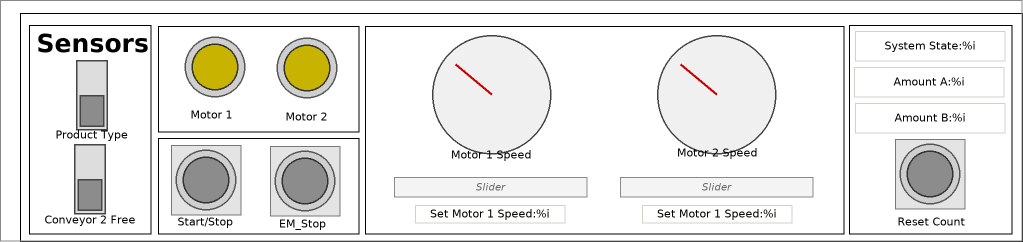
VISUALIZATION Visualization  // 1023x242
    Rectangle (20,13 1003x229)
    Rectangle (849,25 163x209)
    Rectangle (158,138 201x96)
    Rectangle (365,26 479x208)
    Rectangle (158,26 201x106)
    Rectangle (29,25 122x209)
    Lamp1 (180,32 70x70), style: Lamp-Lamp1-Yellow
    Lamp1 (272,33 70x70), variable: GVL.Motor2_State, style: Lamp-Lamp1-Yellow
    DipSwitch (57,60 70x70), variable: GVL.SensorInput, behaviour: TOGGLE, style: Switch-DipSwitch-Gray
    DipSwitch (55,144 70x70), variable: GVL.Conveyor2_Free, behaviour: TOGGLE, style: Switch-DipSwitch-Gray
    Label (18,28 150x30), "Sensors"
    Label (176,100 71x30), "Motor 1"
    Label (271,102 71x30), "Motor 2"
    Meter180 (386,35 211x119), value: GVL.CurrentMotor1_Speed, style: Meter-Meter180-Gray, scale format: %.1f, scale 0..100
    Meter180 (611,35 211x119), value: GVL.CurrentMotor2_Speed, style: Meter-Meter180-Gray, scale format: %.1f, scale 0..100
    Label (430,140 123x30), "Motor 1 Speed"
    Label (656,138 123x30), "Motor 2 Speed"
    Slider (394,177 193x20), variable: GVL.SetMotor1_Speed, scale 0..100
    Slider (620,177 193x20), variable: GVL.SetMotor2_Speed, scale 0..100
    PushSwitchLed (270,146 70x70), variable: GVL.EM_STOP, behaviour: TOGGLE, style: Switch-PushSwitchLed-Gray
    PushSwitch (171,145 70x70), variable: GVL.SART_STOP, behaviour: TOGGLE, style: Switch-PushSwitch-Gray
    Label (170,207 71x30), "Start/Stop"
    Label (267,209 71x30), "EM_Stop"
    Textfield (855,31 150x30), "System State:%i", text variable: GVL.SystemState
    Textfield (415,205 150x18), "Set Motor 1 Speed:%i", text variable: GVL.SetMotor1_Speed
    Textfield (642,205 150x18), "Set Motor 1 Speed:%i", text variable: GVL.SetMotor2_Speed
    Label (41,205 98x30), "Conveyor 2 Free"
    Label (43,120 98x30), "Product Type"
    Textfield (854,67 150x30), "Amount A:%i", text variable: GVL.ProductA_Amount
    Textfield (855,103 150x30), "Amount B:%i", text variable: GVL.ProductB_Amount
    PushSwitch (895,139 70x70), variable: GVL.Reset_Count, behaviour: TOGGLE, style: Switch-PushSwitch-Gray
    Label (870,207 123x30), "Reset Count"
END_VISUALIZATION

(* stored: Version 1.1.0.1, ProductVersion 3.1.4024.12
   Visu Visualization: Id {11180104-6911-46d6-ae10-276ec2a4b535} *)
